Staubli VAL3: start.pgx

program start()
begin
  call Initialisation()
end
